{attribute 'OPC.UA.DA.StructuredType' := '1'}
TYPE ST_FcuControl_out :
STRUCT
	ActForce	: REAL;
	ActPos	: REAL;
	ActWeight	: REAL;
	Contact	: BOOL;
	WeightValid : BOOL;	
	Error	: UINT;
END_STRUCT
END_TYPE

(* stored: Version 1.1.0.1, ProductVersion 3.1.4024.9
   DUT ST_FcuControl_out: Id {e6c17fd3-ba52-4191-8025-634b8a6def0b} *)
